# B&R Automation Studio project DevOpsDemoRepo_Patrick
Automation Studio 6.0.2.177; technology packages: OpcUaCs 6.0.0

## Configuration Config1

CPU 5APC3100.KBU3-000, AutomationRuntime 6.0.2, Build 11.3.0, Vc 6.0.0

### Task classes (Cpu.sw)
```
Cyclic#4:
  Ladder <- Ladder.prg
```

### Hardware
```
5APC3100_KBU3_000 : 5APC3100.KBU3-000 v2.2.7.0
  FileDevice1
  FileDeviceName1 = USER
  FileDevicePath1 = USER_PATH
```

## Logical view

Binary libraries used (declarations not repeated): operator, runtime, AsIecCon, astime, MpAxis, McAxis, MpBase, McBase


### Program Logical/Ladder (IEC)

#### Variables.var
```iecst
VAR
	WorldHello : BOOL;
	HelloWorld : BOOL;
END_VAR
```

#### Cyclic.ld
Diagram, in the editor's own instruction-list form stored in the file:
```il
PROGRAM _CYCLIC

END_PROGRAM
```

Listed in the project but not available here: Logical/Global.typ, Logical/Global.var
